(* PLC project FBD_EVOLUTION_4, Beckhoff Automation GmbH TwinCAT PLC Control 3.5.10.30 *)
(* stored: creationDateTime 2019-09-26T17:06:50.1299821, modificationDateTime 2019-09-26T17:06:50.1299821 *)

PROGRAM POU
VAR
	A: BOOL;
	B: BOOL;
	C: BOOL;
END_VAR
  VAR  (* added by the conversion: wires and edge detectors of the diagram *)
    _EXECUTE10000000004_EN : BOOL;
  END_VAR

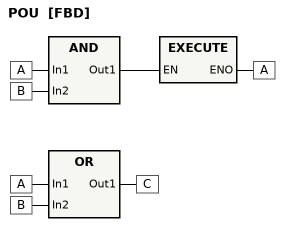
(* FBD diagram, written out as Structured Text *)
_EXECUTE10000000004_EN := A AND B;
IF _EXECUTE10000000004_EN THEN
  A := B;
END_IF;
A := _EXECUTE10000000004_EN;
C := A OR B;
END_PROGRAM

CONFIGURATION Application
  RESOURCE FBD_EVOLUTION_4 ON PLC
(* global variable list GVL *)
{attribute 'qualified_only'}
VAR_GLOBAL
	IsSFCResetting : BOOL;
END_VAR
    TASK PlcTask(INTERVAL := T#0ms, PRIORITY := 20);
    PROGRAM MAIN WITH PlcTask : MAIN;
  END_RESOURCE
END_CONFIGURATION
